Universal Robots PolyScope program: AG SocketComms.urp

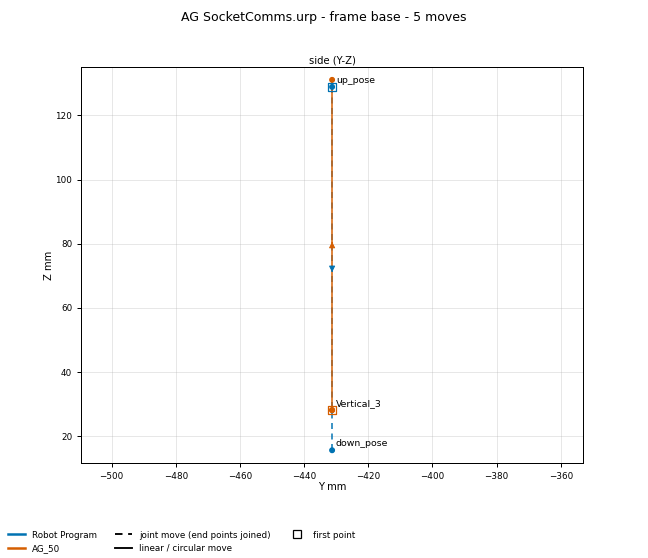
[picture p0: tool path of AG SocketComms.urp in frame base, 5 of 6 moves have a stored position in this frame; points joined in program order, loops and branches not executed]
Program AG SocketComms (installation=default directory=/home/ur/ursim-current/programs createdIn=5.7.0.90932 lastSavedIn=5.9.4.1031232 robotSerialNumber=20195599999)
Calibrated DH parameters: a=[0, -0.425, -0.3922, 0, 0, 0]; d=[0.1625, 0, 0, 0.1333, 0.0997, 0.0996]; alpha=[1.570796, 0, 0, 1.570796, -1.570796, 0]; deltaTheta=[0, 0, 0, 0, 0, 0]
BeforeStart
  start_pose := get_actual_tcp_pose()
  MoveJ speed 60 deg/s, acceleration 80 deg/s^2 (useActiveTCP=true) feature=Base
    Waypoint Waypoint (Variable): variable(name=start_pose)
  Script: socket_close()
  Wait Sleep waitTime=0.25
  socket_is_open := False
  command_index := 0
Robot Program (runOnlyOnce=false)
  Loop While (checkContinuously=false) expression=socket_is_open ≟  False
    socket_is_open := socket_open("192.168.25.1", 30000)
    Wait Sleep waitTime=0.5
  response := "Unknown command"
  command := socket_read_ascii_float(5)
  If command[0]≟5
    Script: socket_send_line("robot_running=True")
    command_index := command_index+1
    Script: socket_set_var("robot_index", command_index)
    Switch expression=command[1]
      Case (caseValue=1)
        MoveL speed 250 mm/s, acceleration 1200 mm/s^2 (useActiveTCP=true) feature=Base
          Waypoint up_pose: TCP in base x=-139.608 y=-431.277 z=128.881 mm, rx=-0.0012 ry=3.1163 rz=0.0389 rad; joints [-91.713, -89.397, -118.352, -63.725, 91.392, -1.776] deg; TCP offset x=0 y=0 z=174 mm, rx=0 ry=0 rz=0 rad
        response := "moved up"
      Case (caseValue=2)
        MoveJ speed 60 deg/s, acceleration 80 deg/s^2 (useActiveTCP=true) feature=Base
          Waypoint down_pose: TCP in base x=-139.608 y=-431.277 z=15.639 mm, rx=-0.0012 ry=3.1163 rz=0.0389 rad; joints [-91.713, -100.473, -126.947, -44.053, 91.392, -1.776] deg
        response := "moved down"
      Case (caseValue=3)
        response := "close"
      Case (caseValue=4)
        response := "open"
      Case (caseValue=50)
        Call AG_50
      Case (caseValue=98)
        response := "socket reset"
      Case (caseValue=99)
        response := "exiting"
      Case (caseValue=2147483647)
        response := "unknown command"
    Script: socket_send_line("robot_response=" + response + "#robot_running=False")
    If command[1]≟98
      Wait Sleep waitTime=0.5
      Script: socket_close()
      socket_is_open := False
    If command[1]≟99
      Wait Sleep waitTime=0.5
      Script: socket_close()
      socket_is_open := False
      Halt
  Else 
    SuppressedNode
      Script: socket_set_var("robot_index", command_index)
SubProgram -> AG_50
SubProgram AG_50 (keepSynchronizedWithDisk=true) programFile=/home/ur/ursim-current/programs/AG_50.urp
  'Rev 2021_12_02am 01'
  MoveL speed 250 mm/s, acceleration 1200 mm/s^2 (useActiveTCP=true) feature=Base
    Waypoint Vertical_3: TCP in base x=-139.608 y=-431.277 z=28.139 mm, rx=-0.0012 ry=3.1163 rz=0.0389 rad; joints [-91.713, -98.956, -126.223, -46.295, 91.392, -1.776] deg
    Waypoint Tilted_1: TCP in base x=-139.608 y=-431.277 z=28.139 mm, rx=-0.0114 ry=3.0194 rz=-0.7761 rad; joints [-92.494, -99.177, -148.291, 6.22, 92.637, -2.25] deg
    Waypoint Vertical_4: TCP in base x=-139.608 y=-431.277 z=131.081 mm, rx=-0.0012 ry=3.1163 rz=0.0389 rad; joints [-91.713, -89.241, -118.143, -64.09, 91.392, -1.776] deg
    response := "50 success"
